FUNCTION_BLOCK EL3102
VAR
	_io : EL3xx2_Data;
	{attribute addProperty Name "WcState"}
	_wcState : WcStateInputToggle;
	{attribute addProperty Name "Info data"}
	_infoData : InfoDataAds;
END_VAR

PROPERTY IO : REFERENCE TO EL3xx2_Data
GET
IO REF= _io;
END_GET
END_PROPERTY

PROPERTY WcState : REFERENCE TO WcStateInputToggle
GET
WcState REF= _wcState;
END_GET
END_PROPERTY

END_FUNCTION_BLOCK

(* stored: Version 1.1.0.1, ProductVersion 3.1.4024.9
   POU EL3102: Id {4877fcee-a287-0501-3d23-6cef2a0aa820}, SpecialFunc None
   Property IO: Id {7754a026-3108-00a7-25e9-6d7b2737ceaf}
   Get Get: Id {36a524b1-9b1f-013c-3fea-a8ff7eb76401}
   Property WcState: Id {f35fd68d-ab8f-00be-00c9-e5eb3bc1ce7e}
   Get Get: Id {b525fd57-2f7a-0407-03ae-e0404cd48793} *)
